(* CoDeSys 2.3.9.35 project: p1q3.pro *)
(* Author: Hemerson *)
(* Libraries: SysLibTargetVisu.lib 26.11.08 09:50:36, Standard.lib 26.11.08 09:46:20, Iecsfc.lib 26.11.08 09:46:14, DU35x.lib 7.7.11 15:59:53, SYSLIBCALLBACK.LIB 26.11.08 09:50:38 *)

(* PLC configuration (modules and I/O channels)
COM1 [COM1] node 0, in %IB0 out %QB0 {BaudRate = 115200; Paridade = No Parity; StopBits = 1 Stop Bit; Modem = Without RTS/CTS; Delay = 5}
  MToolIEC [Codesys] node 0, in %IB0 out %QB0
COM2 [COM2] node 1, in %IB0 out %QB0 {BaudRate = 115200; Paridade = No Parity; StopBits = 1 Stop Bit; Modem = Without RTS/CTS; Delay = 5}
  Disable [Desabilitado485] node 0, in %IB0 out %QB0
I00 AT %IX0.0 [BitInput] I0.0
I01 AT %IX0.1 [BitInput] I0.1
I02 AT %IX0.2 [BitInput] I0.2
I03 AT %IX0.3 [BitInput] I0.3
I04 AT %IX0.4 [BitInput] I0.4
I05 AT %IX0.5 [BitInput] I0.5
I06 AT %IX0.6 [BitInput] I0.6
I07 AT %IX0.7 [BitInput] I0.7
I08 AT %IX0.8 [BitInput] I0.8
Digital Inputs 1 [Entradas1] node 0, in %IW1 out %QB0
  I10 AT %IX1.0 [BitInput] I1.0
  I11 AT %IX1.1 [BitInput] I1.1
  I12 AT %IX1.2 [BitInput] I1.2
  I13 AT %IX1.3 [BitInput] I1.3
  I14 AT %IX1.4 [BitInput] I1.4
  I15 AT %IX1.5 [BitInput] I1.5
  I16 AT %IX1.6 [BitInput] I1.6
  I17 AT %IX1.7 [BitInput] I1.7
  I18 AT %IX1.8 [BitInput] I1.8
Digital Inputs 2 [Entradas2] node 0, in %IW2 out %QB0
  I20 AT %IX2.0 [BitInput] I2.0
  I21 AT %IX2.1 [BitInput] I2.1
Analog Inputs [EntradaAnalogica] node 0, in %IW4 out %QB0
  AI0 AT %IW4 [WordInput] AI0 {TipoAnalogica = Channel Disable; FiltroAnalogica = Filter 0 - AI=2ms  / AV=90ms; FundoEscala = 0}
  AI1 AT %IW5 [WordInput] AI1 {TipoAnalogica = Channel Disable; FiltroAnalogica = Filter 0 - AI=2ms  / AV=90ms; FundoEscala = 0}
  AI2 AT %IW6 [WordInput] AI2 {TipoAnalogica = Channel Disable; FiltroAnalogica = Filter 0 - AI=2ms  / AV=90ms; FundoEscala = 0}
  AI3 AT %IW7 [WordInput] AI3 {TipoAnalogica = Channel Disable; FiltroAnalogica = Filter 0 - AI=2ms  / AV=90ms; FundoEscala = 0}
Fast Inputs [EntradasRapidas] node 1, in %IB16 out %QB0
  Block 0 [Bloco0] node 0, in %IB16 out %QB0
    Disable [DesabilitadoBloco0] node 0, in %IB16 out %QB0
  Block 1 [Bloco1] node 1, in %IB16 out %QB0
    Disable [DesabilitadoBloco1] node 0, in %IB16 out %QB0
  Configurable Input Block 0 [EntradaConfiBloco0] node 2, in %IB16 out %QB0
    Counter 0 [EntradaConfContador0] node 0, in %IB16 out %QB0 {EntradaConfiguravelContador = Disable}
  Configurable Input Block 1 [EntradaConfiBloco1] node 3, in %IB16 out %QB0
    Counter 2 [EntradaConfContador2] node 0, in %IB16 out %QB0 {EntradaConfiguravelContador = Disable}
Q00 AT %QX0.0 [BitOutput] Q0.0
Q01 AT %QX0.1 [BitOutput] Q0.1
Q02 AT %QX0.2 [BitOutput] Q0.2
Q03 AT %QX0.3 [BitOutput] Q0.3
Q04 AT %QX0.4 [BitOutput] Q0.4
Q05 AT %QX0.5 [BitOutput] Q0.5
Q06 AT %QX0.6 [BitOutput] Q0.6
Q07 AT %QX0.7 [BitOutput] Q0.7
Q10 AT %QX1.0 [BitOutput] Q1.0
Q11 AT %QX1.1 [BitOutput] Q1.1
Q12 AT %QX1.2 [BitOutput] Q1.2
Q13 AT %QX1.3 [BitOutput] Q1.3
Q14 AT %QX1.4 [BitOutput] Q1.4
Q15 AT %QX1.5 [BitOutput] Q1.5
Q16 AT %QX1.6 [BitOutput] Q1.6
Q17 AT %QX1.7 [BitOutput] Q1.7
Analog Outputs [SaidaAnalogica] node 0, in %IW0 out %QW3
  AO0 AT %QW3 [WordOutput] AO0 {TipoAnalogica = Channel Disable; FundoEscala = 0}
  AO1 AT %QW4 [WordOutput] AO1 {TipoAnalogica = Channel Disable; FundoEscala = 0}
Fast Outputs [SaidasRapidas] node 1, in %IB0 out %QB10
  Fast Output 0 Disable [DesabilitadoF0] node 0, in %IB0 out %QB10
  Fast Output 1 Disable [DesabilitadoF1] node 1, in %IB0 out %QB10
Counter Output [SaidasContador] node 2, in %IB0 out %QB10
  Block 0 Output Disable [DesabilitadoSaidaBloco0] node 0, in %IB0 out %QB10
  Block 1 Output Disable [DesabilitadoSaidaBloco1] node 1, in %IB0 out %QB10
Timer Event [TimerEvent] node 0, in %IB13 out %QB6 {Intervalo = 10}
*)

(* Global variable list: Variáveis globais *)
VAR_GLOBAL
	TEMPO1: TON;
	TEMPO2: TON;
	TEMPO3: TOF;
	TEMPO4: TON;
	TEMPO5: TOF;
	TEMPO6: TON;
	TEMPO7: TOF;
	TEMPO11: TON;
	TEMPO22: TON;
	TEMPO33: TOF;
	TEMPO44: TON;
	TEMPO55: TOF;
	TEMPO66: TON;
	TEMPO77: TOF;
	OPCOES: CTU;
	Q: BOOL;
	AUX1: BOOL;
	AUX2: BOOL;
	AUX3: BOOL;
	AUX4: BOOL;
	AUX5: BOOL;
	AUX6: BOOL;
	AUX7: BOOL;
	AUX11: BOOL;
	AUX22: BOOL;
	AUX33: BOOL;
	AUX44: BOOL;
	AUX55: BOOL;
	AUX66: BOOL;
	AUX77: BOOL;
	AUXI7: BOOL;
	AUXI0: BOOL;
	CV1: INT;
	CV2: INT;
	S1: BOOL;
	S2: BOOL;
	S3: BOOL;
	S4: BOOL;
	TRIG1: R_TRIG;
	TRIG2: R_TRIG;
	TRIG3: R_TRIG;
	TRIG4: R_TRIG;
	TRIG5: R_TRIG;
	AUXTIME: TIME;
	CONTUD: CTUD;
	RMULT: INT;
	LOAD: BOOL;
	LOAD1: BOOL;
	LOAD2: BOOL;
	OFF: BOOL;
	I0 AT %IX0.0: BOOL;
	I1 AT %IX0.1: BOOL;
	I6 AT %IX0.6: BOOL;
	I7 AT %IX0.7: BOOL;
	O10 AT %QX1.0: BOOL;
	O11 AT %QX1.1: BOOL;
	O12 AT %QX1.2: BOOL;
	O13 AT %QX1.3: BOOL;
	O14 AT %QX1.4: BOOL;
	O15 AT %QX1.5: BOOL;
	O16 AT %QX1.6: BOOL;
	O17 AT %QX1.7: BOOL;
END_VAR

(* POU PLC_PRG, LD *)
PROGRAM PLC_PRG
VAR
	TEMPO1: TON;
	TEMPO2: TON;
	TEMPO3: TOF;
	TEMPO4: TON;
	TEMPO5: TOF;
	TEMPO6: TON;
	TEMPO7: TOF;
	TEMPO11: TON;
	TEMPO22: TON;
	TEMPO33: TOF;
	TEMPO44: TON;
	TEMPO55: TOF;
	TEMPO66: TON;
	TEMPO77: TOF;
	OPCOES: CTU;
	Q: BOOL;
	AUX1: BOOL;
	AUX2: BOOL;
	AUX3: BOOL;
	AUX4: BOOL;
	AUX5: BOOL;
	AUX6: BOOL;
	AUX7: BOOL;
	AUX11: BOOL;
	AUX22: BOOL;
	AUX33: BOOL;
	AUX44: BOOL;
	AUX55: BOOL;
	AUX66: BOOL;
	AUX77: BOOL;
	AUXI7: BOOL;
	AUXI0: BOOL;
	CV1: INT;
	CV2: INT;
	S1: BOOL;
	S2: BOOL;
	S3: BOOL;
	S4: BOOL;
	TRIG1: R_TRIG;
	TRIG2: R_TRIG;
	TRIG3: R_TRIG;
	TRIG4: R_TRIG;
	TRIG5: R_TRIG;
	AUXTIME: TIME;
	CONTUD: CTUD;
	RMULT: INT;
	LOAD: BOOL;
	LOAD1: BOOL;
	LOAD2: BOOL;
	OFF: BOOL;
END_VAR

VAR_INPUT
	I0 AT %IX0.0: BOOL;
	I1 AT %IX0.1: BOOL;
	I6 AT %IX0.6: BOOL;
	I7 AT %IX0.7: BOOL;

END_VAR

VAR_OUTPUT
	O10 AT %QX1.0: BOOL;
	O11 AT %QX1.1: BOOL;
	O12 AT %QX1.2: BOOL;
	O13 AT %QX1.3: BOOL;
	O14 AT %QX1.4: BOOL;
	O15 AT %QX1.5: BOOL;
	O16 AT %QX1.6: BOOL;
	O17 AT %QX1.7: BOOL;
END_VAR
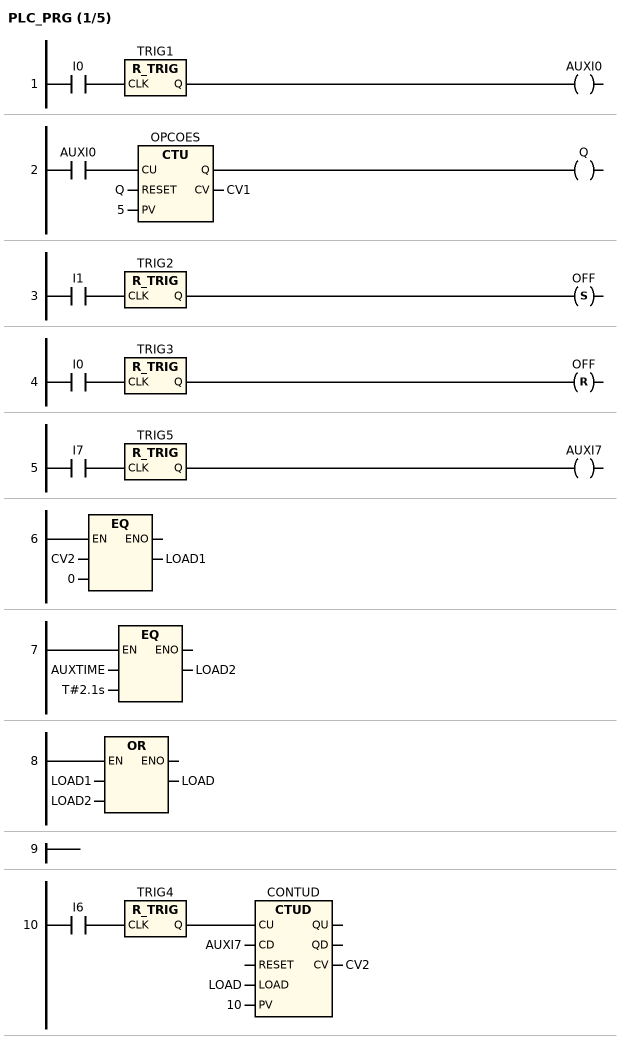
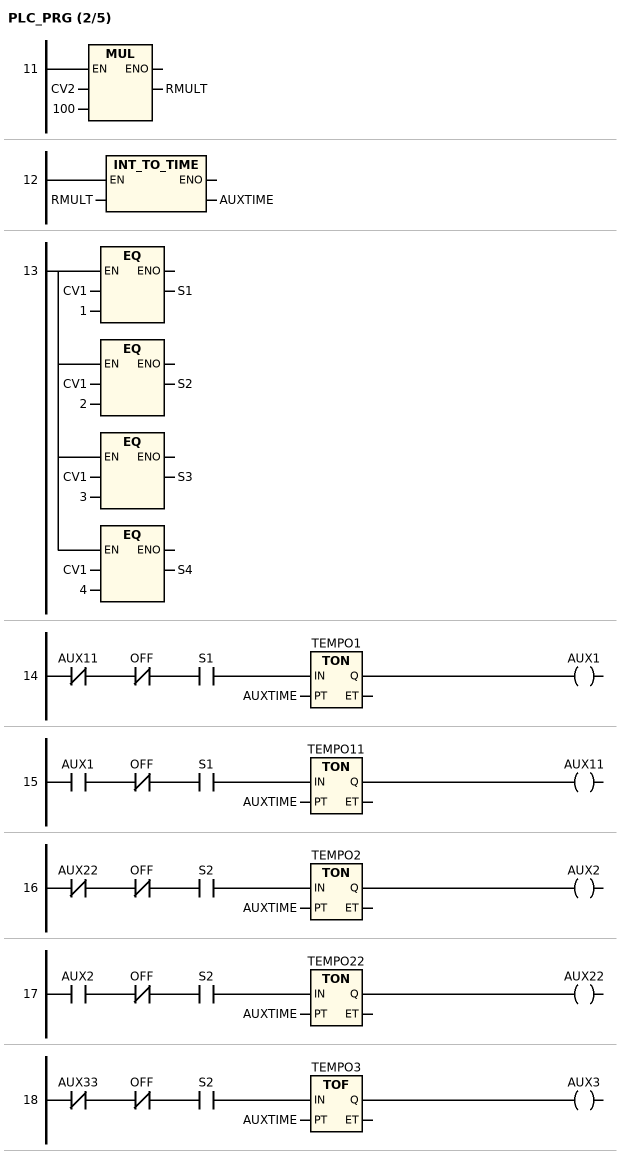
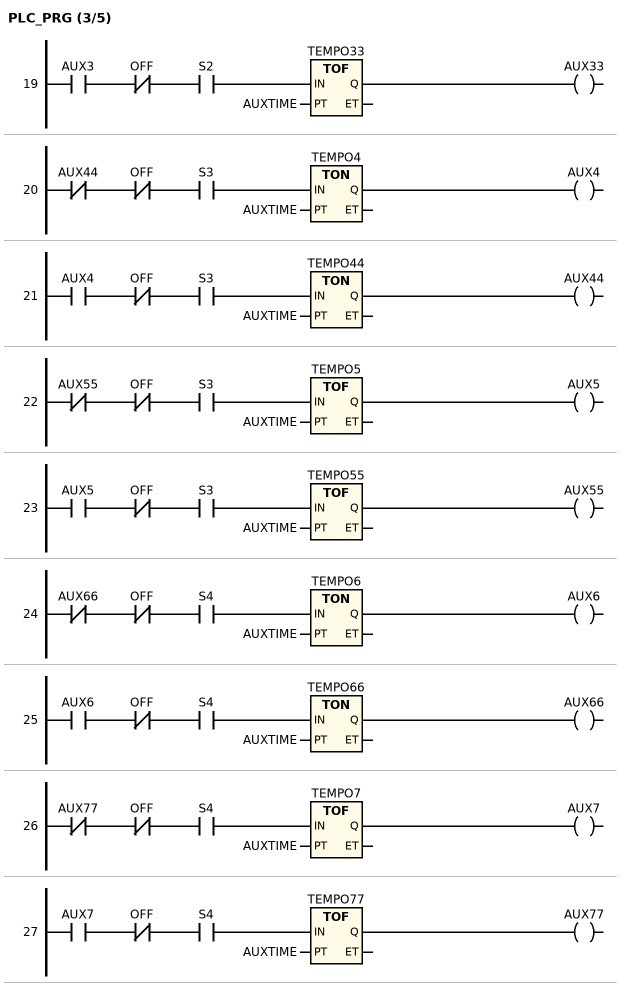
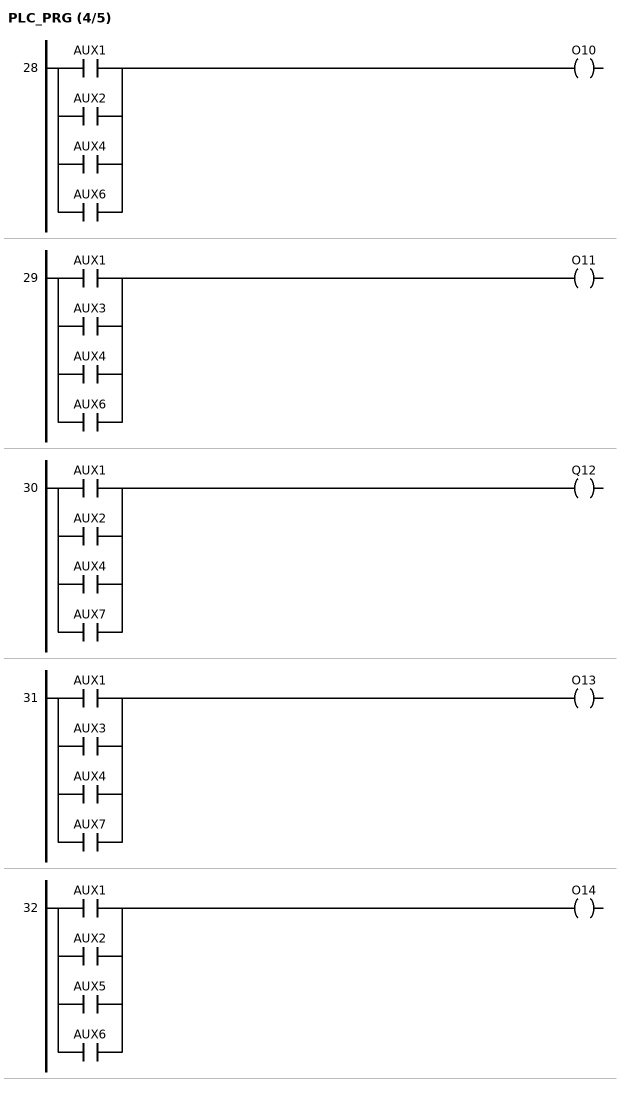
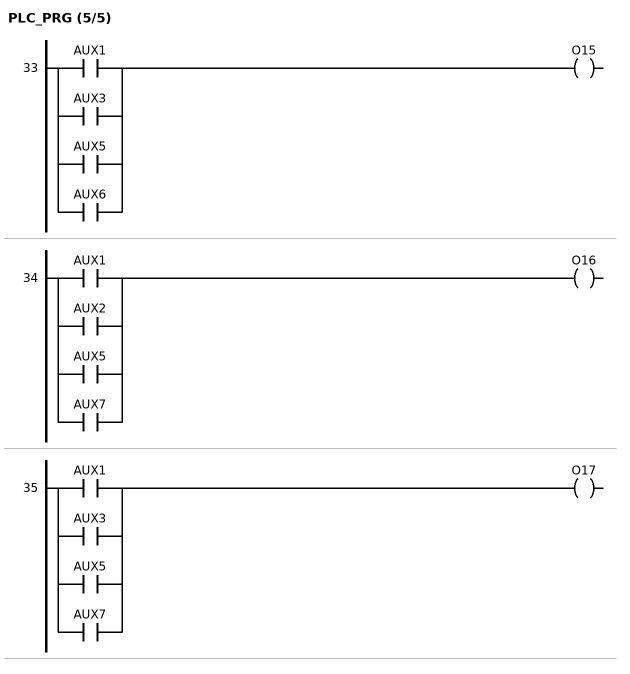
_LD_ (* Ladder Diagram *)
NETWORK 1
	[I0] - TRIG1:R_TRIG(CLK: *) --- (AUXI0)
NETWORK 2
	[AUXI0] - OPCOES:CTU(CU: *, RESET: Q, PV: 5, CV => CV1) --- (Q)
NETWORK 3
	[I1] - TRIG2:R_TRIG(CLK: *) --- (S OFF)
NETWORK 4
	[I0] - TRIG3:R_TRIG(CLK: *) --- (R OFF)
NETWORK 5
	[I7] - TRIG5:R_TRIG(CLK: *) --- (AUXI7)
NETWORK 6
	*
		EN --- EQ(CV2, 0) => LOAD1
NETWORK 7
	*
		EN --- EQ(AUXTIME, T#2.1s) => LOAD2
NETWORK 8
	*
		EN --- OR(LOAD1, LOAD2) => LOAD
NETWORK 9
	*
NETWORK 10
	[I6] - TRIG4:R_TRIG(CLK: *) - CONTUD:CTUD(CU: *, CD: AUXI7, RESET: , LOAD: LOAD, PV: 10, CV => CV2)
NETWORK 11
	*
		EN --- MUL(CV2, 100) => RMULT
NETWORK 12
	*
		EN --- INT_TO_TIME(RMULT) => AUXTIME
NETWORK 13
	*
		EN --- EQ(CV1, 1) => S1
		EN --- EQ(CV1, 2) => S2
		EN --- EQ(CV1, 3) => S3
		EN --- EQ(CV1, 4) => S4
NETWORK 14
	[/AUX11] - [/OFF] - [S1] - TEMPO1:TON(IN: *, PT: AUXTIME) --- (AUX1)
NETWORK 15
	[AUX1] - [/OFF] - [S1] - TEMPO11:TON(IN: *, PT: AUXTIME) --- (AUX11)
NETWORK 16
	[/AUX22] - [/OFF] - [S2] - TEMPO2:TON(IN: *, PT: AUXTIME) --- (AUX2)
NETWORK 17
	[AUX2] - [/OFF] - [S2] - TEMPO22:TON(IN: *, PT: AUXTIME) --- (AUX22)
NETWORK 18
	[/AUX33] - [/OFF] - [S2] - TEMPO3:TOF(IN: *, PT: AUXTIME) --- (AUX3)
NETWORK 19
	[AUX3] - [/OFF] - [S2] - TEMPO33:TOF(IN: *, PT: AUXTIME) --- (AUX33)
NETWORK 20
	[/AUX44] - [/OFF] - [S3] - TEMPO4:TON(IN: *, PT: AUXTIME) --- (AUX4)
NETWORK 21
	[AUX4] - [/OFF] - [S3] - TEMPO44:TON(IN: *, PT: AUXTIME) --- (AUX44)
NETWORK 22
	[/AUX55] - [/OFF] - [S3] - TEMPO5:TOF(IN: *, PT: AUXTIME) --- (AUX5)
NETWORK 23
	[AUX5] - [/OFF] - [S3] - TEMPO55:TOF(IN: *, PT: AUXTIME) --- (AUX55)
NETWORK 24
	[/AUX66] - [/OFF] - [S4] - TEMPO6:TON(IN: *, PT: AUXTIME) --- (AUX6)
NETWORK 25
	[AUX6] - [/OFF] - [S4] - TEMPO66:TON(IN: *, PT: AUXTIME) --- (AUX66)
NETWORK 26
	[/AUX77] - [/OFF] - [S4] - TEMPO7:TOF(IN: *, PT: AUXTIME) --- (AUX7)
NETWORK 27
	[AUX7] - [/OFF] - [S4] - TEMPO77:TOF(IN: *, PT: AUXTIME) --- (AUX77)
NETWORK 28
	{ [AUX1] | [AUX2] | [AUX4] | [AUX6] } --- (O10)
NETWORK 29
	{ [AUX1] | [AUX3] | [AUX4] | [AUX6] } --- (O11)
NETWORK 30
	{ [AUX1] | [AUX2] | [AUX4] | [AUX7] } --- (Q12)
NETWORK 31
	{ [AUX1] | [AUX3] | [AUX4] | [AUX7] } --- (O13)
NETWORK 32
	{ [AUX1] | [AUX2] | [AUX5] | [AUX6] } --- (O14)
NETWORK 33
	{ [AUX1] | [AUX3] | [AUX5] | [AUX6] } --- (O15)
NETWORK 34
	{ [AUX1] | [AUX2] | [AUX5] | [AUX7] } --- (O16)
NETWORK 35
	{ [AUX1] | [AUX3] | [AUX5] | [AUX7] } --- (O17)
_END_LD_
(* the same logic as Structured Text *)
(* Network 1 *)
TRIG1(CLK := I0);
AUXI0 := TRIG1.Q;
(* Network 2 *)
OPCOES(CU := AUXI0, RESET := Q, PV := 5);
CV1 := OPCOES.CV;
Q := OPCOES.Q;
(* Network 3 *)
TRIG2(CLK := I1);
IF TRIG2.Q THEN OFF := TRUE; END_IF;
(* Network 4 *)
TRIG3(CLK := I0);
IF TRIG3.Q THEN OFF := FALSE; END_IF;
(* Network 5 *)
TRIG5(CLK := I7);
AUXI7 := TRIG5.Q;
(* Network 6 *)
LOAD1 := CV2 = 0;
(* Network 7 *)
LOAD2 := AUXTIME = T#2.1s;
(* Network 8 *)
LOAD := LOAD1 OR LOAD2;
(* Network 9: see the listing above *)
(* Network 10: see the listing above *)
(* Network 11 *)
RMULT := CV2 * 100;
(* Network 12 *)
AUXTIME := INT_TO_TIME(RMULT);
(* Network 13 *)
S1 := CV1 = 1;
S2 := CV1 = 2;
S3 := CV1 = 3;
S4 := CV1 = 4;
(* Network 14 *)
TEMPO1(IN := NOT AUX11 AND NOT OFF AND S1, PT := AUXTIME);
AUX1 := TEMPO1.Q;
(* Network 15 *)
TEMPO11(IN := AUX1 AND NOT OFF AND S1, PT := AUXTIME);
AUX11 := TEMPO11.Q;
(* Network 16 *)
TEMPO2(IN := NOT AUX22 AND NOT OFF AND S2, PT := AUXTIME);
AUX2 := TEMPO2.Q;
(* Network 17 *)
TEMPO22(IN := AUX2 AND NOT OFF AND S2, PT := AUXTIME);
AUX22 := TEMPO22.Q;
(* Network 18 *)
TEMPO3(IN := NOT AUX33 AND NOT OFF AND S2, PT := AUXTIME);
AUX3 := TEMPO3.Q;
(* Network 19 *)
TEMPO33(IN := AUX3 AND NOT OFF AND S2, PT := AUXTIME);
AUX33 := TEMPO33.Q;
(* Network 20 *)
TEMPO4(IN := NOT AUX44 AND NOT OFF AND S3, PT := AUXTIME);
AUX4 := TEMPO4.Q;
(* Network 21 *)
TEMPO44(IN := AUX4 AND NOT OFF AND S3, PT := AUXTIME);
AUX44 := TEMPO44.Q;
(* Network 22 *)
TEMPO5(IN := NOT AUX55 AND NOT OFF AND S3, PT := AUXTIME);
AUX5 := TEMPO5.Q;
(* Network 23 *)
TEMPO55(IN := AUX5 AND NOT OFF AND S3, PT := AUXTIME);
AUX55 := TEMPO55.Q;
(* Network 24 *)
TEMPO6(IN := NOT AUX66 AND NOT OFF AND S4, PT := AUXTIME);
AUX6 := TEMPO6.Q;
(* Network 25 *)
TEMPO66(IN := AUX6 AND NOT OFF AND S4, PT := AUXTIME);
AUX66 := TEMPO66.Q;
(* Network 26 *)
TEMPO7(IN := NOT AUX77 AND NOT OFF AND S4, PT := AUXTIME);
AUX7 := TEMPO7.Q;
(* Network 27 *)
TEMPO77(IN := AUX7 AND NOT OFF AND S4, PT := AUXTIME);
AUX77 := TEMPO77.Q;
(* Network 28 *)
O10 := AUX1 OR AUX2 OR AUX4 OR AUX6;
(* Network 29 *)
O11 := AUX1 OR AUX3 OR AUX4 OR AUX6;
(* Network 30 *)
Q12 := AUX1 OR AUX2 OR AUX4 OR AUX7;
(* Network 31 *)
O13 := AUX1 OR AUX3 OR AUX4 OR AUX7;
(* Network 32 *)
O14 := AUX1 OR AUX2 OR AUX5 OR AUX6;
(* Network 33 *)
O15 := AUX1 OR AUX3 OR AUX5 OR AUX6;
(* Network 34 *)
O16 := AUX1 OR AUX2 OR AUX5 OR AUX7;
(* Network 35 *)
O17 := AUX1 OR AUX3 OR AUX5 OR AUX7;
END_PROGRAM

(* Visualisation VP1Q3
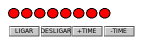
ellipse at (2,2)-(13,12): alarm colour if .O10
ellipse at (15,2)-(26,12): alarm colour if .O11
ellipse at (93,2)-(104,12): alarm colour if .O17
ellipse at (80,2)-(91,12): alarm colour if .O16
ellipse at (28,2)-(39,12): alarm colour if .O12
ellipse at (41,2)-(52,12): alarm colour if .O13
ellipse at (54,2)-(65,12): alarm colour if .O14
ellipse at (67,2)-(78,12): alarm colour if .O15
button at (3,20)-(33,30): text "LIGAR"; toggles .I0
button at (35,20)-(65,30): text "DESLIGAR"; toggles .I1
button at (66,20)-(96,30): text "+TIME"; toggles .I6
button at (98,20)-(128,30): text "-TIME"; toggles .I7
*)
